// TIA Portal V20 export
DATA_BLOCK "DB_Sync"   // DB3
{ S7_Optimized_Access := 'TRUE' }
// stored: MemoryReserve 100
   VAR
      memoryBit : Struct
         System_Byte : Byte;
         FirstScan : Bool;
         DiagStatusUpdate : Bool;
         AlwaysTRUE : Bool;
         AlwaysFALSE : Bool;
      END_STRUCT;
      ClockBit : Struct
         Clock_Byte : Byte;
         Clock_10Hz : Bool;
         Clock_5Hz : Bool;
         "Clock_2.5Hz" : Bool;
         Clock_2Hz : Bool;
         "Clock_1.25Hz" : Bool;
         Clock_1Hz : Bool;
         "Clock_0.625Hz" : Bool;
         "Clock_0.5Hz" : Bool;
      END_STRUCT;
      startbit : Bool;
      stopbit : Bool;
      resetbit : Bool;
   END_VAR
BEGIN
END_DATA_BLOCK
